// TIA Portal V21 export
TYPE "Motor_template"
   STRUCT
      Start : Bool;
      Stop : Bool;
      Status : Bool;
      OverLoad : Bool;
      ShortCircuit : Bool;
      Error1 : Bool;
      Error2 : Bool;
      Error3 : Bool;
      Error4 : Bool;
      Error5 : Bool;
   END_STRUCT;
END_TYPE
